SUBAPPLICATION Uebung_076c_AUI (* MSS mit Compound Scaling + AR_Timeout_Zero auf UT ausgeben (Adapter Version) *)
  (* Standard: 61499-2; Description: Copyright (c) 2026 Meisterschulen am Ostbahnhof This program and the accompanying materials are made available under the terms of the Eclipse Public License 2.0 which is available at https://www.eclipse.org/legal/epl-2.0/ SPDX-License-Identifier: EPL-2.0 *)
  (* Version 1.0, 2026-09-17, Franz Höpfinger, Meisterschulen am Ostbahnhof, MSS mit Compound Scaling und AR_Timeout_Zero SubApp (Adapter Version, analog Krauternter TECU_MSS.SUB) *)
  PACKAGE Uebungen;
  IMPORT Uebungen::const::UT::TECU::DefaultPool_TECU_Numeric::NumberVariable_TECU_Speed_MSS_N;
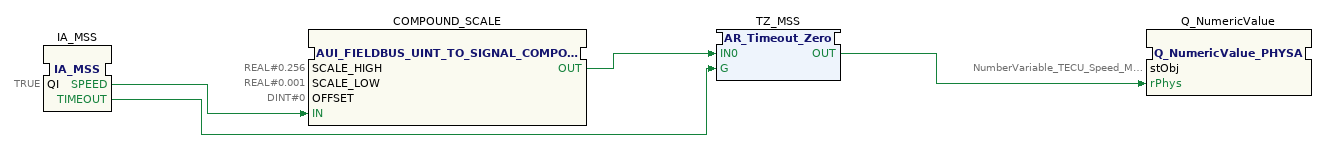
  FBS
    IA_MSS : isobus::tecu::IA_MSS(QI := TRUE);
    COMPOUND_SCALE : logiBUS::signalprocessing::fieldbus::AUI_FIELDBUS_UINT_TO_SIGNAL_COMPOUND_SCALE(SCALE_HIGH := REAL#0.256, SCALE_LOW := REAL#0.001, OFFSET := DINT#0);
    Q_NumericValue : isobus::UT::Q::Q_NumericValue_PHYSA(stObj := NumberVariable_TECU_Speed_MSS_N);
  END_FBS
  SUBAPPS
    TZ_MSS : MyLib::sys::AR_Timeout_Zero;
  END_SUBAPPS
  ADAPTER_CONNECTIONS
    IA_MSS.SPEED TO COMPOUND_SCALE.IN;
    COMPOUND_SCALE.OUT TO TZ_MSS.IN0;
    IA_MSS.TIMEOUT TO TZ_MSS.G;
    TZ_MSS.OUT TO Q_NumericValue.rPhys;
  END_CONNECTIONS
END_SUBAPPLICATION
